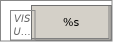
VISUALIZATION VISU_SimpleRelay  // 113x42
VAR_IN_OUT
	ref : SimpleRelay;
    widget : SimpleRelayWidget;
END_VAR
    Button (31,5 80x35), "%s", text variable: widget.text, input disabled if: ref.processes.setEnabled.statuses.enabledStatus.disabled
        OnMouseClick: execute { widget.do_request := TRUE; }
    Frame (10,10 25x30)
        shows VISU_State_gray_green(state := ref.digitalOutput)
END_VISUALIZATION

(* stored: Version 1.1.0.1, ProductVersion 3.1.4019.2
   Visu VISU_SimpleRelay: Id {318d844d-38d2-4587-9c6c-be9f94e0752d} *)
